FUNCTION_BLOCK Crane_PutDownWP EXTENDS Crane_PickPutBase
VAR_INPUT
END_VAR
VAR_OUTPUT
END_VAR
VAR
	m_step: INT := 0;
	m_timer: TON;

	// (EProcessVariables.Crane_HoldingWorkpiece = TRUE) AND (EProcessVariables.Crane_CylinderRetracted = TRUE)
	m_compExpr65: ComparisonExpression(EProcessVariables.Crane_HoldingWorkpiece, EComparisonType.equals, EDataType.binary, TRUE, 0, '', TRUE);
	m_compExpr67: ComparisonExpression(EProcessVariables.Crane_CylinderRetracted, EComparisonType.equals, EDataType.binary, TRUE, 0, '', TRUE);
	m_precondition: BoolExpression(m_compExpr65, EBoolOperation.and_op, m_compExpr67);
	
	// (EProcessVariables.Crane_HoldingWorkpiece = FALSE) AND (EProcessVariables.Crane_CylinderRetracted = TRUE)
	m_compExpr70: ComparisonExpression(EProcessVariables.Crane_HoldingWorkpiece, EComparisonType.equals, EDataType.binary, FALSE, 0, '', TRUE);
	m_compExpr72: ComparisonExpression(EProcessVariables.Crane_CylinderRetracted, EComparisonType.equals, EDataType.binary, TRUE, 0, '', TRUE);
	m_postcondition: BoolExpression(m_compExpr70, EBoolOperation.and_op, m_compExpr72);
END_VAR

SUPER^();

METHOD Abort : BOOL
VAR_INPUT
END_VAR
m_ptrCrane^.o_MonostableCylinder.METH_Retract();
IF m_ptrCrane^.o_VacuumGripper.WPTaken THEN
	m_ptrCrane^.o_VacuumGripper.METH_Intake();
ELSE
	m_ptrCrane^.o_VacuumGripper.METH_Release();
END_IF
Abort := TRUE;
END_METHOD

(* Execution logic of this Control Primitive. *)
METHOD PROTECTED  ExecuteInternal : BOOL
VAR_INPUT
	i_params: ParameterSet;
END_VAR
CASE m_step OF

	0:	// extend
		m_ptrCrane^.o_MonostableCylinder.METH_Extend();
		IF m_ptrCrane^.o_MonostableCylinder.Extended THEN
			m_step := 1;
		END_IF
	
	1:	// release
		m_ptrCrane^.o_VacuumGripper.METH_Release();
		m_timer(IN := TRUE, PT := T#100MS);
		IF m_timer.Q THEN
			m_timer(IN := FALSE);
			m_step := 2;
		END_IF
		
	2: // shift register
		IF ShiftProduct(FALSE) THEN
			m_step := 3;
		END_IF
	
	3:	// retract
		m_ptrCrane^.o_MonostableCylinder.METH_Retract();
		IF m_ptrCrane^.o_MonostableCylinder.Retracted THEN
			m_step := 0;
			ExecuteInternal := TRUE;
		END_IF	
END_CASE
END_METHOD

METHOD FB_init : BOOL
VAR_INPUT
	bInitRetains : BOOL; // if TRUE, the retain variables are initialized (warm start / cold start)
	bInCopyCode : BOOL;  // if TRUE, the instance afterwards gets moved into the copy code (online change)
	
	i_ptrCrane: POINTER TO Crane;
END_VAR
m_ptrCrane := i_ptrCrane;

m_id := EPrimitives.Crane_PutDownWP;
m_timeout := T#20S;

Precondition := m_precondition;
Postcondition := m_postcondition;
END_METHOD

END_FUNCTION_BLOCK

(* stored: Version 1.1.0.1
   POU Crane_PutDownWP: Id {04a27553-468b-4979-8368-e5feadebb203}, SpecialFunc None
   Method Abort: Id {90f6da96-c41b-4844-bf48-1abc163b313d}
   Method ExecuteInternal: Id {e6d71fa5-685c-4df2-8ead-9edbb5f66e4d}
   Method FB_init: Id {ba42f0b9-51e7-4d24-ba8f-ea2205489784} *)
